FUNCTION_BLOCK FB_PowerConveyer
VAR_INPUT
	Enable 		: BOOL;
END_VAR
VAR_OUTPUT
	Status		: BOOL;
	Error		: BOOL;
	Done		: BOOL;
END_VAR
VAR
	fbPower		: MC_Power;
END_VAR

IF Enable THEN
Done := FALSE;
Status := TRUE;
Error := FALSE;


	fbPower(
		Axis := GVL_Conveyer.ConveyerAxis,
		Enable := Enable,
		Enable_Positive := Enable,
		Enable_Negative := Enable,
		);
Status := fbPower.Status;
Error := fbPower.Error;	

IF Status AND NOT Error THEN
	Done := TRUE;
END_IF

END_IF

END_FUNCTION_BLOCK

(* stored: Version 1.1.0.1, ProductVersion 3.1.4024.11
   POU FB_PowerConveyer: Id {6c662a5d-d672-4b4d-99fd-36c3d8f8bd1f}, SpecialFunc None *)
